Universal Robots PolyScope program: grab_egg.urp

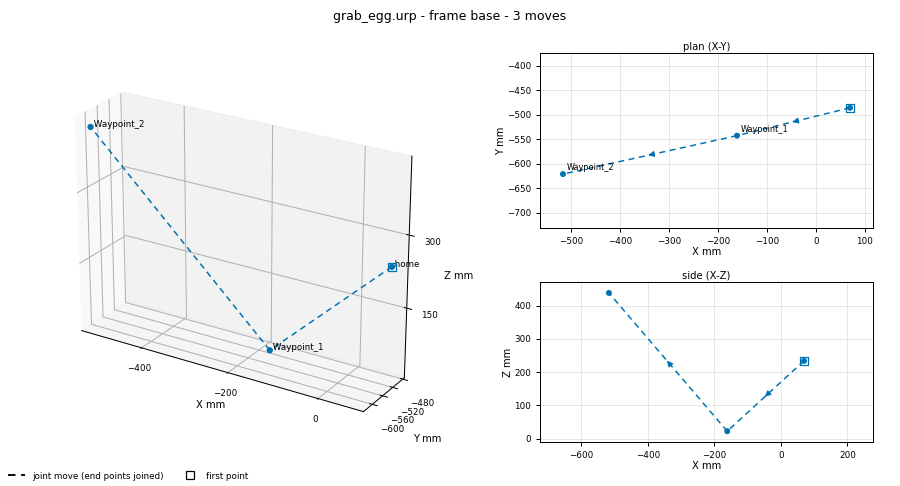
[picture p0: tool path of grab_egg.urp in frame base, 3 of 3 moves have a stored position in this frame; points joined in program order, loops and branches not executed]
Program grab_egg (installation=default directory=/programs/usbdisk/brazo_final/grab_egg createdIn=5.13.0 lastSavedIn=5.13.0 robotSerialNumber=20205500280)
Calibrated DH parameters: a=[0.000126, -0.227628, -0.392536, 0.000072, 0.000053, 0]; d=[0.16267, 78.773992, -78.210517, -0.430145, 0.099656, 0.099678]; alpha=[1.568545, -0.004566, 0.00572, 1.569931, -1.57104, 0]; deltaTheta=[0, -1.006608, 7.298003, -0.008206, 0.000004, 0]
InitVariablesNode
Robot Program (runOnlyOnce=false)
  MoveJ speed 60 deg/s, acceleration 80 deg/s^2 (useActiveTCP=true) feature=Base
    Waypoint home: TCP in base x=69.599 y=-485.817 z=233.686 mm, rx=2.0537 ry=-2.3377 rz=-0.0319 rad; joints [83.686, -92.519, 95.471, -93.426, -91.591, 91.281] deg; TCP offset x=0 y=0 z=234.35 mm, rx=0 ry=0 rz=-3.1416 rad
    URCap RG6 (RG - On Robot, OnRobot A/S) dataModel(depthCompensate=false, force=120, payload=0.0, width=90, name=RG6(90))
  MoveJ speed 60 deg/s, acceleration 80 deg/s^2 (useActiveTCP=true) feature=Base
    Waypoint Waypoint_1: TCP in base x=-161.372 y=-542.767 z=22.22 mm, rx=-2.2363 ry=-2.1897 rz=-0.0088 rad; joints [59.999, -72.994, 105.66, -122.184, -90.243, -118.369] deg; TCP offset x=0 y=0 z=234.35 mm, rx=0 ry=0 rz=-3.1416 rad
    URCap RG6 (RG - On Robot, OnRobot A/S) dataModel(force=120, payload=0.0, depthCompensate=true, width=32, name=RG6(32))
  MoveJ speed 60 deg/s, acceleration 80 deg/s^2 (useActiveTCP=true) feature=Base
    Waypoint Waypoint_2: TCP in base x=-516.94 y=-621.246 z=437.883 mm, rx=1.9579 ry=0.4178 rz=-1.7518 rad; joints [46.309, -70.766, 101.831, -206.949, -104.142, -80.244] deg; TCP offset x=0 y=0 z=234.35 mm, rx=0 ry=0 rz=-3.1416 rad
